PROGRAM MAIN
VAR
	Input1 AT %I* : BOOL ;
	Output1 AT %Q* : BOOL ;
END_VAR

Output1 := Input1;

SafetyLogic();

Gvl_Var.EthOB0.1 := FlashBits.Bits.3;
Gvl_Var.EthOB0.2 := FlashBits.Bits.4;

END_PROGRAM

(* stored: Version 1.1.0.1, ProductVersion 3.1.4026.8
   POU MAIN: Id {97141ba4-d654-40f7-b7ee-9901641685db}, SpecialFunc None *)
